TYPE eXML :
	(	
		OK,
		errMaxBufferLen,
		errStringLen,
		Error
	);
END_TYPE

(* stored: Version 1.1.0.1, ProductVersion 3.1.4022.18
   DUT eXML: Id {05a4fdda-1086-47b5-ad10-7c2bac568355} *)
